// TIA Portal V16 export
// export: Created 2022-09-01T14:26:55.6358864Z, ExportSetting WithDefaults, DisplayName Totally Integrated Automation Portal, DisplayVersion V16, DisplayName TIA Portal Version Control Interface, DisplayVersion V16, DisplayName TIA Portal Openness, DisplayVersion V16, DisplayName STEP 7 Professional, DisplayVersion V16, DisplayName STEP 7 Safety, DisplayVersion V16, DisplayName WinCC Advanced, DisplayVersion V16
FUNCTION "UV" : Void   // FC15, LAD
{ S7_Optimized_Access := 'TRUE' }
VERSION : 0.1
// stored: AutoNumber true, IsIECCheckEnabled false, SetENOAutomatically false, UDAEnableTagReadback false
   VAR_TEMP
      sr_ultravioleta : Bool;
   END_VAR
BEGIN

REGION Network 1
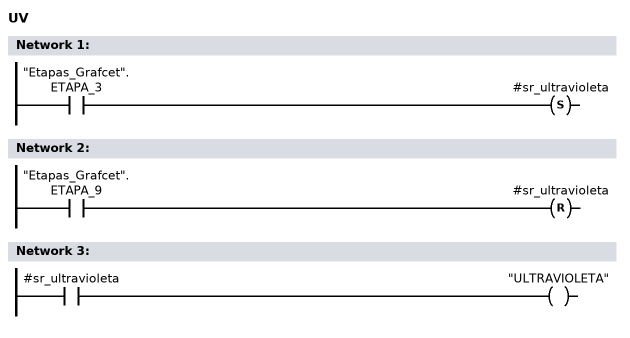
   RUNG wire#powerrail
      Contact( "Etapas_Grafcet".ETAPA_3 )
      S_Coil( #sr_ultravioleta )
   END_RUNG
   // the same network as SCL:
   IF "Etapas_Grafcet".ETAPA_3 THEN #sr_ultravioleta := TRUE; END_IF;
END_REGION

REGION Network 2
   RUNG wire#powerrail
      Contact( "Etapas_Grafcet".ETAPA_9 )
      R_Coil( #sr_ultravioleta )
   END_RUNG
   // the same network as SCL:
   IF "Etapas_Grafcet".ETAPA_9 THEN #sr_ultravioleta := FALSE; END_IF;
END_REGION

REGION Network 3
   RUNG wire#powerrail
      Contact( #sr_ultravioleta )
      Coil( "ULTRAVIOLETA" )
   END_RUNG
   // the same network as SCL:
   "ULTRAVIOLETA" := #sr_ultravioleta;
END_REGION
END_FUNCTION
